// TIA Portal project "Sortierer" (V20)

(* hardware
DEVICE "S7-300/ET200M-Station_1"  S7-300 station
   slot 0: "Profilschiene_0"  Rail  6ES7 390-1***0-0AA0
   slot 2: "PLC_1"  CPU 315-2 PN/DP  6ES7 315-2EH14-0AB0  V3.2.18
      slot 2: "PROFINET-Schnittstelle_1"  PN-IO
         slot 1: "Port_1"  Port
         slot 2: "Port_2"  Port
   slot 4: "DI 16x24VDC_1"  DI16 x 24VDC, interrupt  6ES7 321-7BH01-0AB0
   slot 5: "DO 16x24VDC/0.5A_1"  DO16 x 24VDC / 0.5A  6ES7 322-1BH01-0AA0
*)

// ===== PLC "PLC_1"  CPU 315-2 PN/DP =====

VAR_GLOBAL   // PLC tag table "Standard-Variablentabelle"
   "Förderband_an" AT %M1.2 : Bool;
   "Förderband_aus" AT %M1.3 : Bool;
   "NotAus_aktiv" AT %M1.1 : Bool;
   "Takt_100Hz" AT %M100.5 : Bool;
   "Anlage_ein" AT %M1.0 : Bool;
   "Paket_erkannt" AT %M2.2 : Bool;
   "Paket_klein" AT %M2.0 : Bool;
   "Paket_gross" AT %M2.1 : Bool;
   "Kolben_aktiv" AT %M3.0 : Bool;
   "Kolben_inaktiv" AT %M3.1 : Bool;
   "Förderband_freigeben" AT %M2.5 : Bool;
   "Förderband_stoppen" AT %M2.4 : Bool;
   "Tag_1" AT %M0.0 : Bool;
   "Tag_2" AT %M0.1 : Bool;
END_VAR

VAR_GLOBAL   // PLC tag table "Eingänge"
   "S1" AT %E0.4 : Bool;   // Start-Taster
   "S2" AT %E0.5 : Bool;   // Stopp-Taster
   "S4" AT %E0.0 : Bool;   // Not-Aus Schalter
   "S0" AT %E0.1 : Bool;   // Betriebsschalter auf ein
   "S3" AT %E0.6 : Bool;   // Rücksetz-Taster
   "1B1_S" AT %E1.0 : Bool;   // Hinterer Kolben-Sensor
   "2B1_S" AT %E1.1 : Bool;   // Vorderer Kolben-Sensor
   "S5" AT %E1.3 : Bool;   // Sensor Lichttaster am Kolben
   "1S1_S" AT %E1.4 : Bool;   // Lichtschranke (Strahl 3)
   "2S1_S" AT %E1.5 : Bool;   // Lichtschranke (Strahl 2)
   "3S1_S" AT %E1.6 : Bool;   // Lichtschranke (Strahl 1)
   "4S1_S" AT %E1.7 : Bool;   // Lichtschranke (Strahl 0)
END_VAR

VAR_GLOBAL   // PLC tag table "Ausgänge"
   "S1_Licht" AT %A0.4 : Bool;   // Lampe des Start-Tasters
   "S2_Licht" AT %A0.5 : Bool;   // Lampe des Stopp-Tasters
   "M1" AT %A0.0 : Bool;   // Förderband
   "S3_Licht" AT %A0.6 : Bool;   // Lampe des Rücksetz-Tasters
   "H1" AT %A0.1 : Bool;   // Meldeleuchte (Grün)
   "H2" AT %A0.2 : Bool;   // Meldeleuchte (Gelb)
   "H3" AT %A0.3 : Bool;   // Meldeleuchte (Rot)
   "1M1" AT %A1.0 : Bool;   // Kolbensteuerung
END_VAR

FUNCTION "Paketbandanlage" : Void   // FC1, FBD
{ S7_Optimized_Access := 'FALSE' }
VERSION : 0.1
   VAR_TEMP   // added for the SCL form of the ladder/FBD networks
      _w1 : Bool;
   END_VAR
BEGIN

REGION Network 1: Paketbandsteuerung
   // Hinweis: Alle Schalter können nur benutzt werden, wenn die Anlage über den Betriebsschalter eingeschaltet wurde.
   // Das Paketband kann dann über S1 (Start-Taster) eingeschaltet werden und läuft dann dauerhaft. Über S2 (Stopp-Taster) kann das Paketband ausgeschaltet werden. Der Stopp-Modus, kann über durch den Start deaktiviert werden.
   // Beide Modi (Start, Stopp) werden deaktiviert, sobald S4 (Not-Aus Schalter) aktiv ist.
   // Der Not-Aus-Modus kann nur über S3 (Rücksetz-Taster) deaktiviert werden.
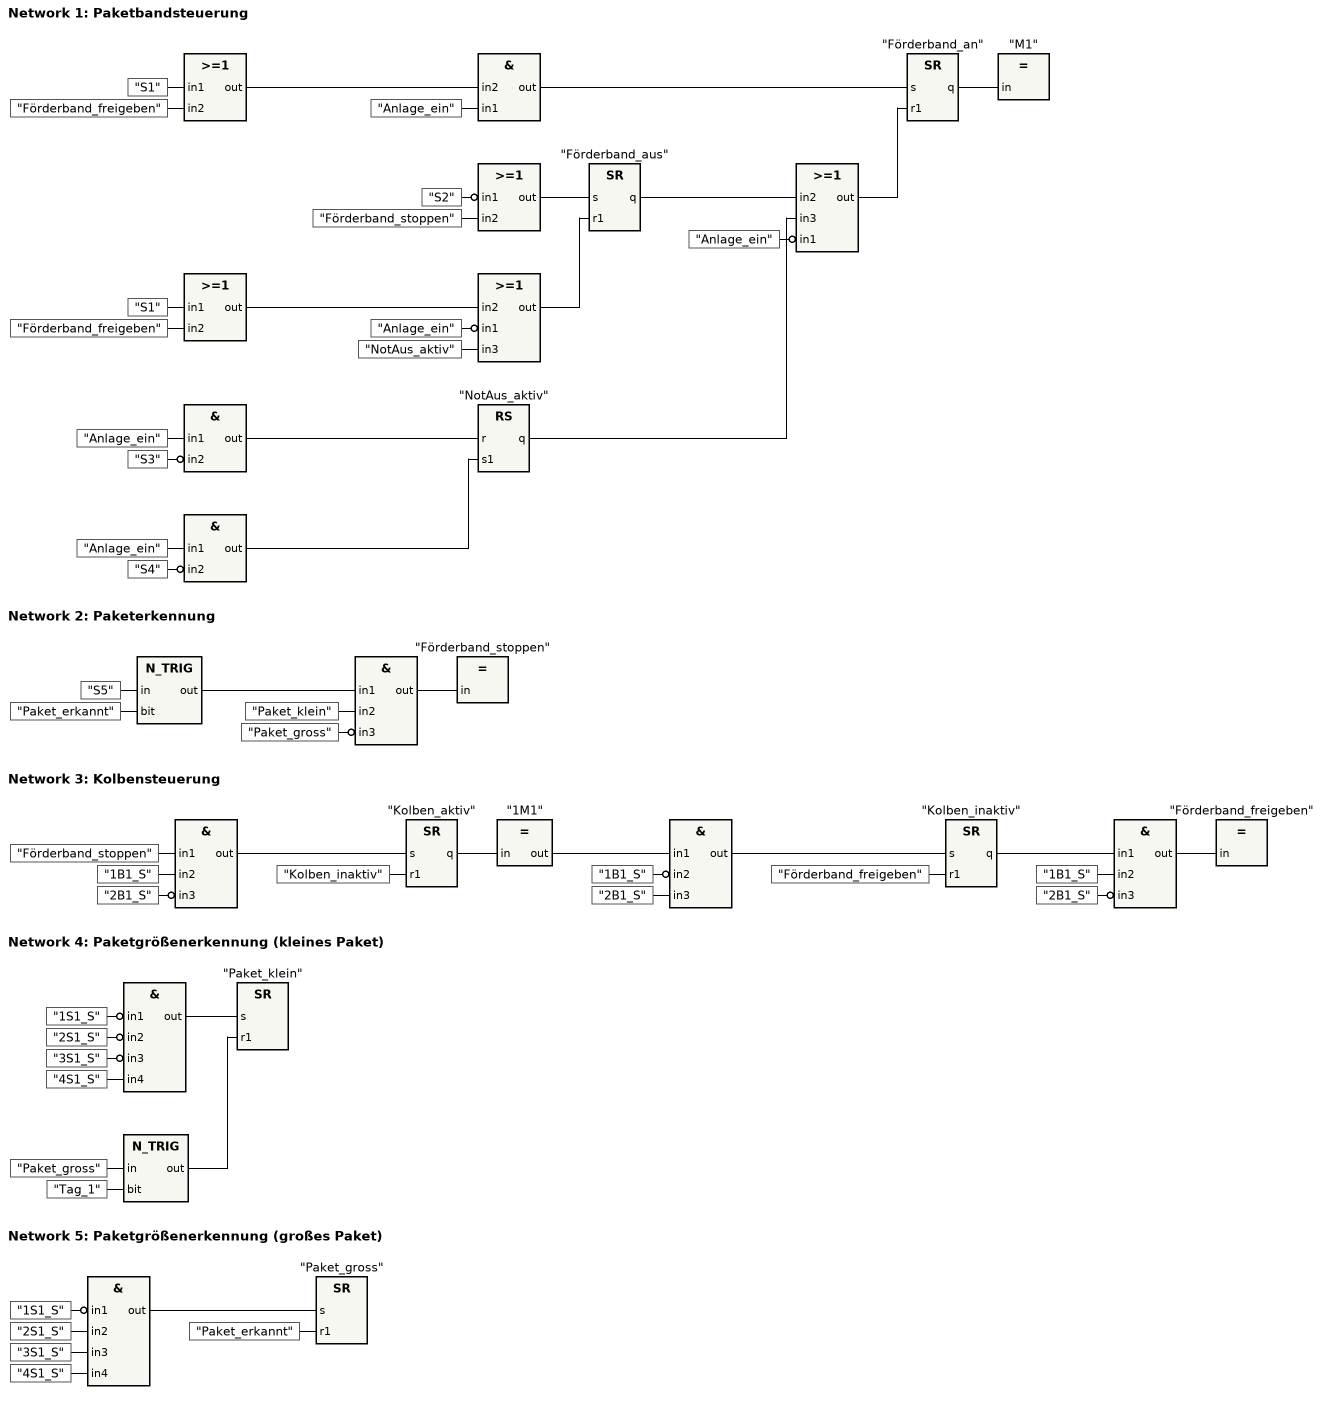
   IF NOT "S2" OR "Förderband_stoppen" THEN
       "Förderband_aus" := TRUE;   // SR flip-flop
   END_IF;
   IF "S1" OR "Förderband_freigeben" OR NOT "Anlage_ein" OR "NotAus_aktiv" THEN
       "Förderband_aus" := FALSE;
   END_IF;
   IF "Anlage_ein" AND NOT "S3" THEN
       "NotAus_aktiv" := FALSE;   // RS flip-flop
   END_IF;
   IF "Anlage_ein" AND NOT "S4" THEN "NotAus_aktiv" := TRUE; END_IF;
   IF ("S1" OR "Förderband_freigeben") AND "Anlage_ein" THEN
       "Förderband_an" := TRUE;   // SR flip-flop
   END_IF;
   IF "Förderband_aus" OR "NotAus_aktiv" OR NOT "Anlage_ein" THEN "Förderband_an" := FALSE; END_IF;
   "M1" := "Förderband_an";
END_REGION

REGION Network 2: Paketerkennung
   // Wenn ein Paket erkannt wird und es sich um ein kleines Paket handelt, dann wird das Förderband gestoppt. Andernfalls soll das Förderband weiterlaufen.
   #_w1 := NOT "S5" AND "Paket_erkannt";   // falling edge
   "Paket_erkannt" := "S5";
   "Förderband_stoppen" := #_w1 AND "Paket_klein" AND NOT "Paket_gross";
END_REGION

REGION Network 3: Kolbensteuerung
   // Nachdem das Förderband gestoppt wurde (kleines Paket liegt vor dem Schieber), wird der Kolben aus- und wieder eingefahren. Danach wird das Förderband wieder freigegeben.
   IF "Förderband_stoppen" AND "1B1_S" AND NOT "2B1_S" THEN
       "Kolben_aktiv" := TRUE;   // SR flip-flop
   END_IF;
   IF "Kolben_inaktiv" THEN "Kolben_aktiv" := FALSE; END_IF;
   "1M1" := "Kolben_aktiv";
   IF "Kolben_aktiv" AND NOT "1B1_S" AND "2B1_S" THEN
       "Kolben_inaktiv" := TRUE;   // SR flip-flop
   END_IF;
   IF "Förderband_freigeben" THEN "Kolben_inaktiv" := FALSE; END_IF;
   "Förderband_freigeben" := "Kolben_inaktiv" AND "1B1_S" AND NOT "2B1_S";
END_REGION

REGION Network 4: Paketgrößenerkennung (kleines Paket)
   // Hier wird getestet, ob es sich um ein kleines Paket handelt. Dazu darf nur der untere Sensor der Lichtschranke aktiv sein. Wir nehmen an, dass die Pakete immer klein sind, bis ein großes Paket den Zustand zurück setzt.
   #_w1 := NOT "Paket_gross" AND "Tag_1";   // falling edge
   "Tag_1" := "Paket_gross";
   IF NOT "1S1_S" AND NOT "2S1_S" AND NOT "3S1_S" AND "4S1_S" THEN
       "Paket_klein" := TRUE;   // SR flip-flop
   END_IF;
   IF #_w1 THEN "Paket_klein" := FALSE; END_IF;
END_REGION

REGION Network 5: Paketgrößenerkennung (großes Paket)
   // Hier wird getestet, ob es sich um ein großes Paket handelt. Dazu dürfen nur die unteren drei Sensoren der Lichtschranke aktiv sein. Wenn ein neues Paket erkannt wird, werden die Daten zurück gesetzt.
   IF NOT "1S1_S" AND "2S1_S" AND "3S1_S" AND "4S1_S" THEN
       "Paket_gross" := TRUE;   // SR flip-flop
   END_IF;
   IF "Paket_erkannt" THEN "Paket_gross" := FALSE; END_IF;
END_REGION

REGION Network 6: Leuchtensteuerung (Aktiv)
   // Wenn die Anlage ein ist und gestartet wurde, dann soll die Meldeleuchte und die Leuchte des Start-Tasters leuchten.
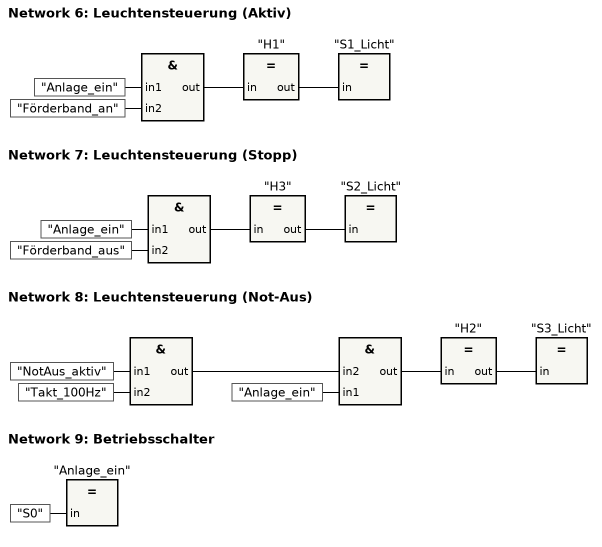
   "H1" := "Anlage_ein" AND "Förderband_an";
   "S1_Licht" := "H1";
END_REGION

REGION Network 7: Leuchtensteuerung (Stopp)
   // Wenn die Anlage ein ist, aber gestoppt wurde, dann soll die Meldeleuchte und die Leuchte des Stopp-Tasters leuchten.
   "H3" := "Anlage_ein" AND "Förderband_aus";
   "S2_Licht" := "H3";
END_REGION

REGION Network 8: Leuchtensteuerung (Not-Aus)
   // Wenn die Anlage ein ist und sich im Not-Aus befindet, dann soll die Meldeleuchte und die Leuchte des Rücksetz-Tasters blinken.
   "H2" := "NotAus_aktiv" AND "Takt_100Hz" AND "Anlage_ein";
   "S3_Licht" := "H2";
END_REGION

REGION Network 9: Betriebsschalter
   // Wenn der Betriebsschalter auf ein steht, sollen bestimmte Funktionsweisen möglich sein.
   "Anlage_ein" := "S0";
END_REGION
END_FUNCTION

ORGANIZATION_BLOCK "Main"   // OB1, FBD
TITLE = "Main Program Sweep (Cycle)"
{ S7_Optimized_Access := 'FALSE' }
VERSION : 0.1
   VAR_TEMP
      OB1_EV_CLASS : Byte;   // Bits 0-3 = 1 (Coming event), Bits 4-7 = 1 (Event class 1)
      OB1_SCAN_1 : Byte;   // 1 (Cold restart scan 1 of OB 1), 3 (Scan 2-n of OB 1)
      OB1_PRIORITY : Byte;   // Priority of OB Execution
      OB1_OB_NUMBR : Byte;   // 1 (Organization block 1, OB1)
      OB1_RESERVED_1 : Byte;   // Reserved for system
      OB1_RESERVED_2 : Byte;   // Reserved for system
      OB1_PREV_CYCLE : Int;   // Cycle time of previous OB1 scan (milliseconds)
      OB1_MIN_CYCLE : Int;   // Minimum cycle time of OB1 (milliseconds)
      OB1_MAX_CYCLE : Int;   // Maximum cycle time of OB1 (milliseconds)
      OB1_DATE_TIME : Date_And_Time;   // Date and time OB1 started
   END_VAR
BEGIN

REGION Network 1
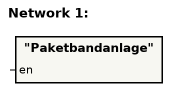
   "Paketbandanlage"();
END_REGION
END_ORGANIZATION_BLOCK